// TIA Portal V17 program export: 1 tag tables, 0 data types, 2 data blocks, 5 code blocks (in call order from the OBs), 0 instance data blocks

VAR_GLOBAL   // PLC tag table "Default tag table"
   Tag_1 AT %M0.0 : Bool;
   Tag_2 AT %M0.1 : Bool;
END_VAR

DATA_BLOCK "FBD_Block_DB"
{ S7_Optimized_Access := 'TRUE' }
VERSION : 0.1
NON_RETAIN
"FBD_Block"

BEGIN

END_DATA_BLOCK

DATA_BLOCK "SCL_Block_DB"
{ S7_Optimized_Access := 'TRUE' }
VERSION : 0.1
NON_RETAIN
"SCL_Block"

BEGIN

END_DATA_BLOCK

ORGANIZATION_BLOCK "Main"   // OB1, LAD, ProgramCycle
TITLE = "Main Program Sweep (Cycle)"
{ S7_Optimized_Access := 'TRUE' }
VERSION : 0.1
// stored: AutoNumber true, IsIECCheckEnabled false, SetENOAutomatically false
   VAR_INPUT
      Initial_Call : Bool;   // Initial call of this OB
      Remanence : Bool;   // =True, if remanent data are available
   END_VAR
   VAR_TEMP   // added for the SCL form of the ladder/FBD networks
      _w1 : Bool;
   END_VAR
BEGIN

REGION Network 1
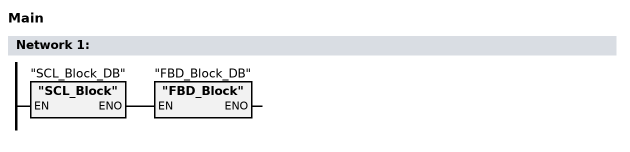
   RUNG wire#powerrail
      "SCL_Block_DB"()
      "FBD_Block_DB"()
   END_RUNG
   // the same network as SCL:
   "SCL_Block_DB"(ENO => #_w1);   // "SCL_Block"
   IF #_w1 THEN
       "FBD_Block_DB"();   // "FBD_Block"
   END_IF;
END_REGION
END_ORGANIZATION_BLOCK

FUNCTION_BLOCK "SCL_Block"
{ S7_Optimized_Access := 'TRUE' }
VERSION : 0.1
   VAR 
      statCondition : Bool;
      aa : Int;
   END_VAR


BEGIN
	IF #statCondition = TRUE THEN
	    // Statement section IF
	    
	    ;
	END_IF;
	FOR #aa:=1 TO 10 DO
	    // Statement section FOR
	    ;
	END_FOR;
	
	
	
END_FUNCTION_BLOCK

FUNCTION_BLOCK "FBD_Block"   // FB2, FBD
{ S7_Optimized_Access := 'TRUE' }
VERSION : 0.1
// stored: AutoNumber true, IsIECCheckEnabled false, IsRetainMemResEnabled false, MemoryReserve 100, SetENOAutomatically false, UDAEnableTagReadback false
   VAR
      statInfo : Word := 16#5;
      statInfo2 : Word;
   END_VAR
BEGIN

REGION Network 1
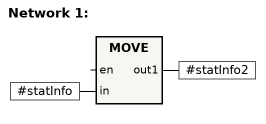
   #statInfo2 := #statInfo;
END_REGION
END_FUNCTION_BLOCK

FUNCTION_BLOCK "Block_1"   // FB3, LAD
{ S7_Optimized_Access := 'TRUE' }
VERSION : 0.1
// stored: AutoNumber true, IsIECCheckEnabled false, IsRetainMemResEnabled false, MemoryReserve 100, SetENOAutomatically false, UDAEnableTagReadback false
   VAR_INPUT
      "a" : Bool;
   END_VAR
   VAR_OUTPUT
      "b" : Bool;
   END_VAR
   VAR_IN_OUT
      c : Bool;
   END_VAR
   VAR
      d : Bool;
   END_VAR
   VAR_TEMP
      "e" : Bool;
   END_VAR
   VAR CONSTANT
      f : Bool;
   END_VAR
BEGIN

REGION Network 1
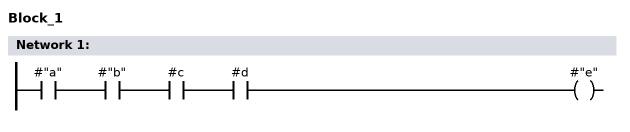
   RUNG wire#powerrail
      Contact( #"a" )
      Contact( #"b" )
      Contact( #c )
      Contact( #d )
      Coil( #"e" )
   END_RUNG
   // the same network as SCL:
   #"e" := #"a" AND #"b" AND #c AND #d;
END_REGION
END_FUNCTION_BLOCK

FUNCTION "Block_2" : Void   // FC1, LAD
{ S7_Optimized_Access := 'TRUE' }
VERSION : 0.1
// stored: AutoNumber true, IsIECCheckEnabled false, SetENOAutomatically false, UDAEnableTagReadback false
BEGIN

REGION Network 1
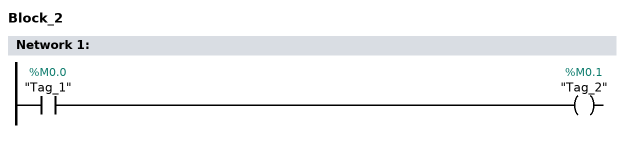
   RUNG wire#powerrail
      Contact( "Tag_1" )
      Coil( "Tag_2" )
   END_RUNG
   // the same network as SCL:
   "Tag_2" := "Tag_1";
END_REGION
END_FUNCTION
